(* PLC project RetentiveDemo, Soft PLC Simulator Retentive Fixture 1.0 *)
(* stored: creationDateTime 2026-07-22T00:00:00, modificationDateTime 2026-07-22T00:00:00 *)

PROGRAM Main
  VAR RETAIN
    Accumulator : DINT := 0;
  END_VAR
  VAR
    Scratch : INT;
  END_VAR

Accumulator := Accumulator + 1;
END_PROGRAM

CONFIGURATION Config0
  RESOURCE Res0 ON PLC
    VAR_GLOBAL RETAIN
      TotalCount : DINT := 0;
      LastRecipe : STRING;
    END_VAR
    VAR_GLOBAL
      Heartbeat : BOOL;
    END_VAR
    VAR_GLOBAL CONSTANT
      MaxTemp : REAL := 150.0;
    END_VAR
  END_RESOURCE
END_CONFIGURATION
